RoboDK station: Proyecto Juan Hector2 (1).rdk

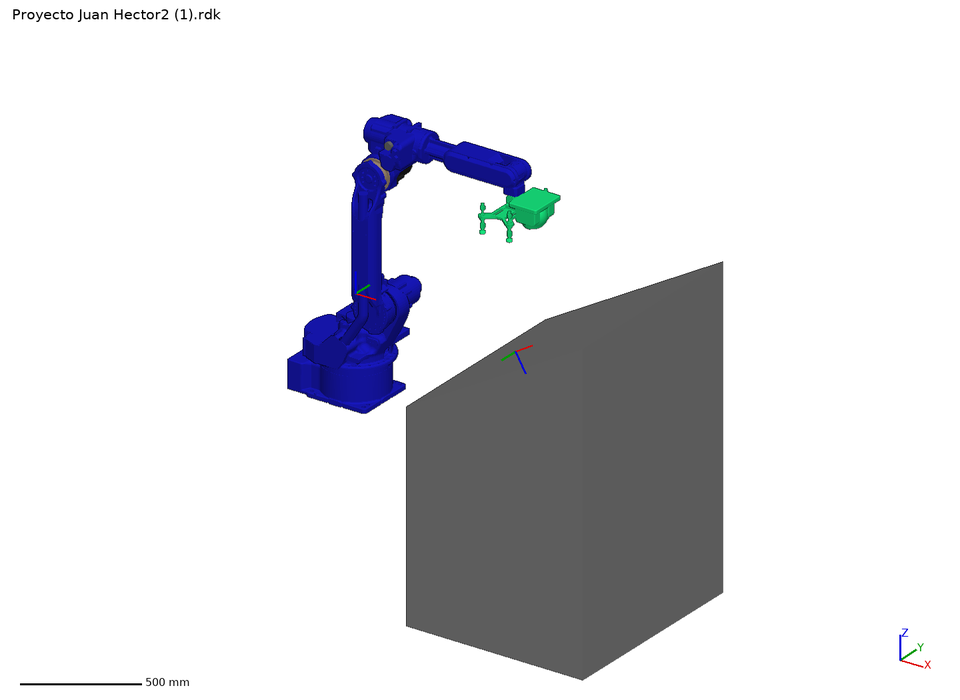
[picture v0: the station drawn from its stored meshes, robots at their saved joint values, targets as dots, program paths as lines]
Station Proyecto Juan Hector2 (saved by RoboDK 5.9.1). Poses are relative to the parent item; angles as X-Y-Z fixed-axis rotations.
  - frame Motoman MH6 Base at (0, 0, 450) mm
    - robot Motoman MH6: 6 axes, payload 6 kg, reach 1422 mm, repeatability 0.08 mm, weight 130 kg
        modified DH rows (alpha deg, a mm, theta deg, d mm): 0, 0, 0, 450; -90, 152, -90, 0; 0, 614, 0, 0; -90, 155, 0, 640; 90, 0, 90, 0; -90, 0, 0, 95
        base shift (0, 0, -450) mm
        joint limits [-170, -90, -175, -180, -45, -360] to [170, 155, 250, 180, 225, 360]; home [0, 0, 0, 0, 0, 0]; saved at [0, 0, 0, 0, 0, 0]
      - tool Ventosas, TCP at (0, 0, 190) mm, size 250 x 290 x 148 mm
    - frame Frame_from_Target1 at (823.2, -34.49, -21.13) mm, rotated rx -180 ry -30 rz 0 deg
  - object CAJA2 at (1600, 500, 300) mm, rotated rx 180 ry 0 rz 0 deg, size 886.4 x 1000 x 1511.7 mm, geometry from CAJA2.stp
  - Python program RosPolar (listed below)

--- Python program RosPolar ---
from robodk.robolink import *
from robodk.robomath import *
import math

#------------------------------------------------
# 1) Conexión e inicialización
#------------------------------------------------
RDK = Robolink()

#Elegir un robot (si hay varios, aparece un popup)
robot = RDK.ItemUserPick("Selecciona un robot", ITEM_TYPE_ROBOT)
if not robot.Valid():
    raise Exception("No se ha seleccionado un robot válido.")
print("Robot conectado correctamente.")

# Conectar al robot físico
#if not robot.Connect():
    #raise Exception("No se pudo conectar al robot. Verifica que esté en modo remoto y que la configuración sea correcta.")

# Confirmar conexión
#if not robot.ConnectedState():
    #raise Exception("El robot no está conectado correctamente. Revisa la conexión.")

#print("Robot conectado correctamente.")

#------------------------------------------------
# 2) Frame de referencia
#------------------------------------------------
frame_name = "Frame_from_Target1"
frame = RDK.Item(frame_name, ITEM_TYPE_FRAME)
if not frame.Valid():
    raise Exception(f'No se encontró el Frame "{frame_name}".')

robot.setPoseFrame(frame)
robot.setPoseTool(robot.PoseTool())
robot.setSpeed(300)
robot.setRounding(5)

#------------------------------------------------
# 3) Parámetros
#------------------------------------------------
z_surface = 0
z_safe = 50
scale = 1.5
spacing = 35 * scale


#------------------------------------------------
# 4) Movimiento al centro en altura segura
#------------------------------------------------

home_pose = robot.Pose()


# El centro de la rosa (r=0) corresponde a x=0, y=0
robot.MoveJ(transl(0, 0, z_surface + z_safe))

# Bajamos a la "superficie" (Z=0)
robot.MoveL(transl(0, 0, z_surface))


#------------------------------------------------
# 4) Funciones de letras
#------------------------------------------------
def draw_letter(points):
    x0, y0 = points[0]
    robot.MoveJ(transl(x0, y0, z_surface + z_safe))
    robot.MoveL(transl(x0, y0, z_surface))
    for (x, y) in points:
        robot.MoveL(transl(x, y, z_surface))
    robot.MoveL(transl(x, y, z_surface + z_safe))

def draw_J(xo, yo):
    points = []
    r = 15 * scale
    for i in range(20):
        angle = math.pi * i / 19
        x = r * math.cos(angle)
        y = r * math.sin(angle)
        points.append((x, y))
    height = 80 * scale
    for i in range(10):
        x = 0
        y = r + i * (height / 9)
        points.append((x, y))
    points.append((10 * scale, r + height))
    return [(xo + x, yo + y) for (x, y) in points]

def draw_U(xo, yo):
    points = []
    r = 15 * scale
    height = 80 * scale
    for i in range(10):
        x = -r
        y = i * height / 9
        points.append((x, y))
    for i in range(20):
        angle = math.pi - (math.pi * i / 19)
        x = r * math.cos(angle)
        y = height + r * math.sin(angle)
        points.append((x, y))
    for i in range(10):
        x = r
        y = height - i * height / 9
        points.append((x, y))
    return [(xo + x, yo + y) for (x, y) in points]

def draw_A(xo, yo):
    w = 30 * scale
    h = 80 * scale
    points = [
        (0, 0), (-w/2, h), (0, h - 10*scale), (w/2, h), (0, 0),
        (-w/4, h/2), (w/4, h/2)
    ]
    return [(xo + x, yo + y) for (x, y) in points]

def draw_N(xo, yo):
    w = 30 * scale
    h = 80 * scale
    points = [(0, 0), (0, h), (w, 0), (w, h)]
    return [(xo + x, yo + y) for (x, y) in points]

def draw_H(xo, yo):
    w = 30 * scale
    h = 80 * scale
    points = [(0, 0), (0, h), (0, h/2), (w, h/2), (w, 0), (w, h)]
    return [(xo + x, yo + y) for (x, y) in points]

def draw_E(xo, yo):
    w = 30 * scale
    h = 80 * scale
    points = [(w, h), (0, h), (0, 0), (w, 0), (0, 0), (0, h/2), (w*0.6, h/2)]
    return [(xo + x, yo + y) for (x, y) in points]

def draw_C(xo, yo):
    r = 30 * scale
    h = 80 * scale
    cx = 0
    cy = h/2
    points = []
    for i in range(30):
        angle = math.pi/4 + math.pi * i / 29
        x = cx + r * math.cos(angle)
        y = cy + r * math.sin(angle)
        points.append((xo + x, yo + y))
    return points

def draw_T(xo, yo):
    w = 30 * scale
    h = 80 * scale
    points = [(w/2, 0), (w/2, h), (0, h), (w, h)]
    return [(xo + x, yo + y) for (x, y) in points]

def draw_O(xo, yo):
    r = 30 * scale
    h = 80 * scale
    cx = 0
    cy = h/2
    points = []
    for i in range(40):
        angle = 2 * math.pi * i / 39
        x = cx + r * math.cos(angle)
        y = cy + r * math.sin(angle)
        points.append((xo + x, yo + y))
    return points

def draw_R(xo, yo):
    h = 80 * scale
    r = 15 * scale
    w = 30 * scale
    points = [(0, 0), (0, h), (0, h*0.6)]
    for i in range(20):
        angle = math.pi * i / 19
        x = r * math.cos(angle)
        y = h*0.6 + r * math.sin(angle)
        points.append((x, y))
    points.append((0, h*0.6))
    points.append((w, 0))
    return [(xo + x, yo + y) for (x, y) in points]


  # ── Emoji tipo "smiley" (☺) usando coordenadas polares ─────────
def draw_face(xo, yo):
    """
    Dibuja una carita feliz:
        • Círculo principal
        • Dos ojos (círculos pequeños)
        • Sonrisa (arco)
    Todo generado con r=f(θ) para trayectorias suaves.
    """
    # Tamaños relativos
    face_r      = 40 * scale          # radio de la cara
    eye_r       = 5  * scale          # radio de cada ojo
    eye_offset  = 15 * scale          # desplazamiento de los ojos
    mouth_r     = 20 * scale          # radio del arco de la boca
    mouth_drop  = 10                  # cuán “abajo” va la sonrisa

    # 1) Contorno circular de la cara
    face_pts = [(xo + face_r*math.cos(t),
                 yo + face_r*math.sin(t))
                for t in [2*math.pi*i/99 for i in range(100)]]
    draw_letter(face_pts)

    # 2) Ojo izquierdo
    left_eye = [(xo - eye_offset + eye_r*math.cos(t),
                 yo + eye_offset + eye_r*math.sin(t))
                for t in [2*math.pi*i/19 for i in range(20)]]
    draw_letter(left_eye)

    # 3) Ojo derecho
    right_eye = [(xo + eye_offset + eye_r*math.cos(t),
                  yo + eye_offset + eye_r*math.sin(t))
                 for t in [2*math.pi*i/19 for i in range(20)]]
    draw_letter(right_eye)

    # 4) Sonrisa – solo medio‐arco inferior
    smile = [(xo + mouth_r*math.cos(t),
              yo - mouth_drop + mouth_r*math.sin(t))
             for t in [math.pi*i/29 for i in range(30)]]
    draw_letter(smile)


#------------------------------------------------
# 5) Dibujo de las palabras
#------------------------------------------------

origin_x = 0
origin_y = 0

# Palabra JUAN
draw_letter(draw_J(origin_x + 0 * spacing, origin_y))
draw_letter(draw_U(origin_x + 1 * spacing, origin_y))
draw_letter(draw_A(origin_x + 2 * spacing, origin_y))
draw_letter(draw_N(origin_x + 3 * spacing, origin_y))

# Palabra HECTOR (en segunda línea o más a la derecha)
offset_x = origin_x + 5.5 * spacing
draw_letter(draw_H(offset_x + 0 * spacing, origin_y))
draw_letter(draw_E(offset_x + 1 * spacing, origin_y))
draw_letter(draw_C(offset_x + 2 * spacing, origin_y))
draw_letter(draw_T(offset_x + 3 * spacing, origin_y))
draw_letter(draw_O(offset_x + 4 * spacing, origin_y))
draw_letter(draw_R(offset_x + 5 * spacing, origin_y))

print("¡Palabras 'JUAN HECTOR' dibujadas correctamente!")

# Emoji (-_-) debajo de las letras
emoji_x = origin_x + 3 * spacing
emoji_y = origin_y - 100  # Más abajo
draw_face(emoji_x, emoji_y)

# Volver al target "Home" si existe
robot.MoveJ(home_pose)
